Staubli VAL3: util.pjx

--- util.pjx ---
Parameters version=s7.6 stackSize=5000 millimeterUnit=true
Program file=_decode.pgx
Program file=_getVersion.pgx
Program file=_str2Array.pgx
Program file=_toString.pgx
Program file=_trsf2String.pgx
Program file=addNumToString.pgx
Program file=addStrToString.pgx
Program file=binToDec.pgx
Program file=bmask.pgx
Program file=BuildString.pgx
Program file=centerCircle.pgx
Program file=COM.pgx
Program file=decToBin.pgx
Program file=extractPos.pgx
Program file=fillStr.pgx
Program file=getLibName.pgx
Program file=isBitSet.pgx
Program file=padding.pgx
Program file=setBit.pgx
Program file=SHL.pgx
Program file=SHR.pgx
Program file=start.pgx
Program file=stop.pgx
Program file=strAlign.pgx
Program file=uSpy.pgx
Data file=util.dtx

--- DECTOBIN.pgx ---
public program decToBin(num x_value, string& x_return[])
// change num variable to binary string (e.g. 9 => "1001")
  local num l_bit
  local num l_value
  local num l_mask
begin
  l_mask=0
  l_bit=1
  x_return=""
  l_value=roundDown(x_value)
  do
    call bmask(l_bit,l_mask)
    if (l_value%2)==0
      x_return="0"+x_return
    else
      x_return="1"+x_return
    endIf
    l_value=roundDown(l_value/2)
    l_bit=l_bit+1
  until l_mask>x_value
  if bDebug
    putln("decToBin(): "+toString("0.0",x_value)+" => "+x_return)
  endIf
end
